// TIA Portal V18 export
FUNCTION "Status" : Void   // FC27, LAD
{ S7_Optimized_Access := 'TRUE' }
VERSION : 0.1
// stored: AutoNumber true, IsIECCheckEnabled false, SetENOAutomatically false, UDAEnableTagReadback false
BEGIN

REGION Network 1: Drive control A nok
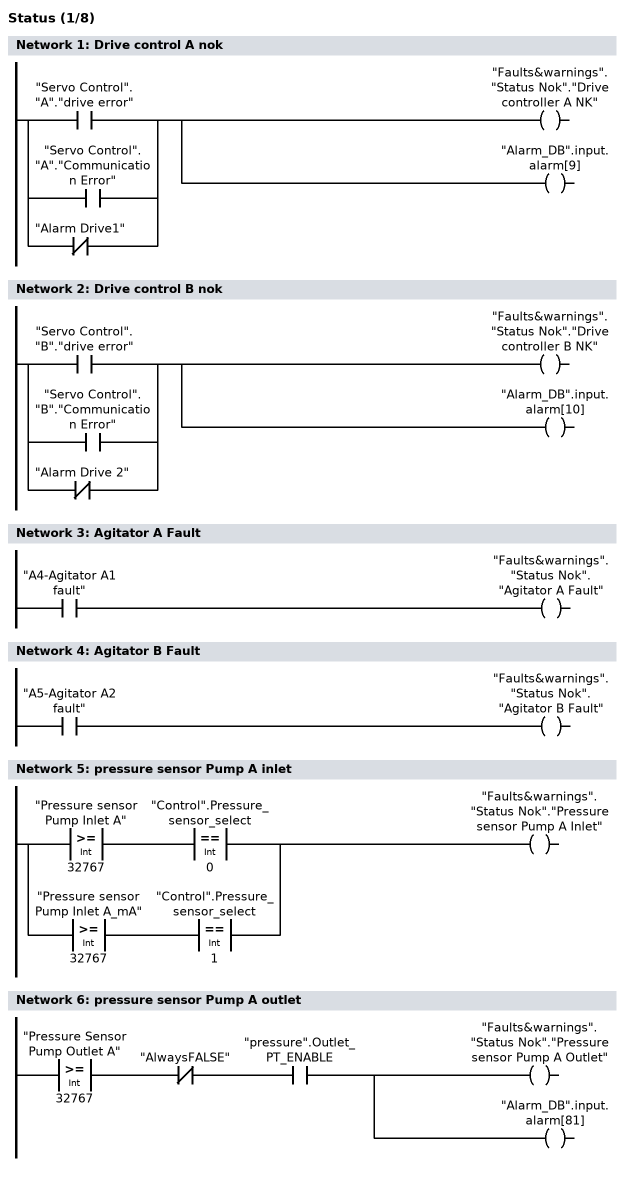
   RUNG wire#powerrail
      Contact( "Servo Control"."A"."drive error" )
      wire#w1
      Coil( "Faults&warnings"."Status Nok"."Drive controller A NK" )
   END_RUNG
   RUNG wire#powerrail
      Contact( "Servo Control"."A"."Communication Error" )
   END_RUNG wire#w1
   RUNG wire#powerrail
      I_Contact( "Alarm Drive1" )
   END_RUNG wire#w1
   RUNG wire#w1
      Coil( "Alarm_DB".input.alarm[9] )
   END_RUNG
   // the same network as SCL:
   "Faults&warnings"."Status Nok"."Drive controller A NK" := "Servo Control"."A"."drive error" OR "Servo Control"."A"."Communication Error" OR NOT "Alarm Drive1";
   "Alarm_DB".input.alarm[9] := "Faults&warnings"."Status Nok"."Drive controller A NK";
END_REGION

REGION Network 2: Drive control B nok
   RUNG wire#powerrail
      Contact( "Servo Control"."B"."drive error" )
      wire#w1
      Coil( "Faults&warnings"."Status Nok"."Drive controller B NK" )
   END_RUNG
   RUNG wire#powerrail
      Contact( "Servo Control"."B"."Communication Error" )
   END_RUNG wire#w1
   RUNG wire#powerrail
      I_Contact( "Alarm Drive 2" )
   END_RUNG wire#w1
   RUNG wire#w1
      Coil( "Alarm_DB".input.alarm[10] )
   END_RUNG
   // the same network as SCL:
   "Faults&warnings"."Status Nok"."Drive controller B NK" := "Servo Control"."B"."drive error" OR "Servo Control"."B"."Communication Error" OR NOT "Alarm Drive 2";
   "Alarm_DB".input.alarm[10] := "Faults&warnings"."Status Nok"."Drive controller B NK";
END_REGION

REGION Network 3: Agitator A Fault
   RUNG wire#powerrail
      Contact( "A4-Agitator A1 fault" )
      Coil( "Faults&warnings"."Status Nok"."Agitator A Fault" )
   END_RUNG
   // the same network as SCL:
   "Faults&warnings"."Status Nok"."Agitator A Fault" := "A4-Agitator A1 fault";
END_REGION

REGION Network 4: Agitator B Fault
   RUNG wire#powerrail
      Contact( "A5-Agitator A2 fault" )
      Coil( "Faults&warnings"."Status Nok"."Agitator B Fault" )
   END_RUNG
   // the same network as SCL:
   "Faults&warnings"."Status Nok"."Agitator B Fault" := "A5-Agitator A2 fault";
END_REGION

REGION Network 5: pressure sensor Pump A inlet
   RUNG wire#powerrail
      { S7_Templates := "SrcType := Int" } GE_Contact(in1 := "Pressure sensor Pump Inlet A", in2 := 32767)
      { S7_Templates := "SrcType := Int" } EQ_Contact(in1 := "Control".Pressure_sensor_select, in2 := 0)
      wire#w1
      Coil( "Faults&warnings"."Status Nok"."Pressure sensor Pump A Inlet" )
   END_RUNG
   RUNG wire#powerrail
      { S7_Templates := "SrcType := Int" } GE_Contact(in1 := "Pressure sensor Pump Inlet A_mA", in2 := 32767)
      { S7_Templates := "SrcType := Int" } EQ_Contact(in1 := "Control".Pressure_sensor_select, in2 := 1)
   END_RUNG wire#w1
   // the same network as SCL:
   "Faults&warnings"."Status Nok"."Pressure sensor Pump A Inlet" := (("Pressure sensor Pump Inlet A" >= 32767) AND ("Control".Pressure_sensor_select = 0)) OR (("Pressure sensor Pump Inlet A_mA" >= 32767) AND ("Control".Pressure_sensor_select = 1));
END_REGION

REGION Network 6: pressure sensor Pump A outlet
   RUNG wire#powerrail
      { S7_Templates := "SrcType := Int" } GE_Contact(in1 := "Pressure Sensor Pump Outlet A", in2 := 32767)
      I_Contact( "AlwaysFALSE" )
      Contact( "pressure".Outlet_PT_ENABLE )
      wire#w1
      Coil( "Faults&warnings"."Status Nok"."Pressure sensor Pump A Outlet" )
   END_RUNG
   RUNG wire#w1
      Coil( "Alarm_DB".input.alarm[81] )
   END_RUNG
   // the same network as SCL:
   "Faults&warnings"."Status Nok"."Pressure sensor Pump A Outlet" := ("Pressure Sensor Pump Outlet A" >= 32767) AND NOT "AlwaysFALSE" AND "pressure".Outlet_PT_ENABLE;
   "Alarm_DB".input.alarm[81] := "Faults&warnings"."Status Nok"."Pressure sensor Pump A Outlet";
END_REGION

REGION Network 7: pressure sensor Pump B inlet
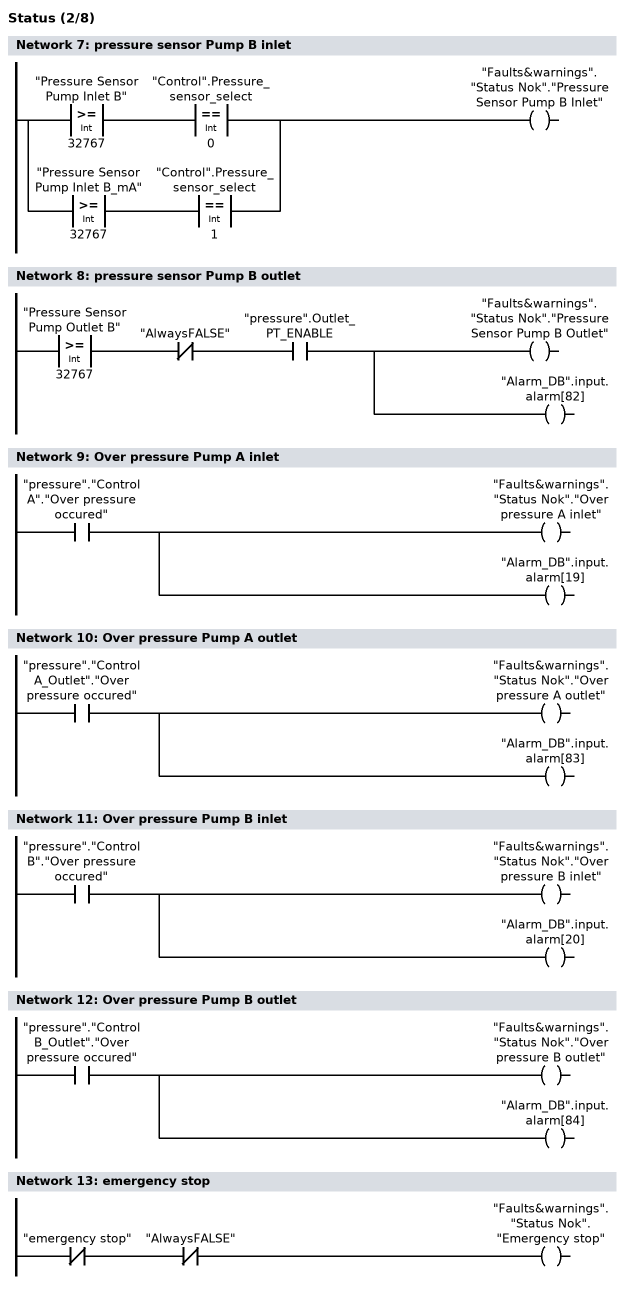
   RUNG wire#powerrail
      { S7_Templates := "SrcType := Int" } GE_Contact(in1 := "Pressure Sensor Pump Inlet B", in2 := 32767)
      { S7_Templates := "SrcType := Int" } EQ_Contact(in1 := "Control".Pressure_sensor_select, in2 := 0)
      wire#w1
      Coil( "Faults&warnings"."Status Nok"."Pressure Sensor Pump B Inlet" )
   END_RUNG
   RUNG wire#powerrail
      { S7_Templates := "SrcType := Int" } GE_Contact(in1 := "Pressure Sensor Pump Inlet B_mA", in2 := 32767)
      { S7_Templates := "SrcType := Int" } EQ_Contact(in1 := "Control".Pressure_sensor_select, in2 := 1)
   END_RUNG wire#w1
   // the same network as SCL:
   "Faults&warnings"."Status Nok"."Pressure Sensor Pump B Inlet" := (("Pressure Sensor Pump Inlet B" >= 32767) AND ("Control".Pressure_sensor_select = 0)) OR (("Pressure Sensor Pump Inlet B_mA" >= 32767) AND ("Control".Pressure_sensor_select = 1));
END_REGION

REGION Network 8: pressure sensor Pump B outlet
   RUNG wire#powerrail
      { S7_Templates := "SrcType := Int" } GE_Contact(in1 := "Pressure Sensor Pump Outlet B", in2 := 32767)
      I_Contact( "AlwaysFALSE" )
      Contact( "pressure".Outlet_PT_ENABLE )
      wire#w1
      Coil( "Faults&warnings"."Status Nok"."Pressure Sensor Pump B Outlet" )
   END_RUNG
   RUNG wire#w1
      Coil( "Alarm_DB".input.alarm[82] )
   END_RUNG
   // the same network as SCL:
   "Faults&warnings"."Status Nok"."Pressure Sensor Pump B Outlet" := ("Pressure Sensor Pump Outlet B" >= 32767) AND NOT "AlwaysFALSE" AND "pressure".Outlet_PT_ENABLE;
   "Alarm_DB".input.alarm[82] := "Faults&warnings"."Status Nok"."Pressure Sensor Pump B Outlet";
END_REGION

REGION Network 9: Over pressure Pump A inlet
   RUNG wire#powerrail
      Contact( "pressure"."Control A"."Over pressure occured" )
      wire#w1
      Coil( "Faults&warnings"."Status Nok"."Over pressure A inlet" )
   END_RUNG
   RUNG wire#w1
      Coil( "Alarm_DB".input.alarm[19] )
   END_RUNG
   // the same network as SCL:
   "Faults&warnings"."Status Nok"."Over pressure A inlet" := "pressure"."Control A"."Over pressure occured";
   "Alarm_DB".input.alarm[19] := "pressure"."Control A"."Over pressure occured";
END_REGION

REGION Network 10: Over pressure Pump A outlet
   RUNG wire#powerrail
      Contact( "pressure"."Control A_Outlet"."Over pressure occured" )
      wire#w1
      Coil( "Faults&warnings"."Status Nok"."Over pressure A outlet" )
   END_RUNG
   RUNG wire#w1
      Coil( "Alarm_DB".input.alarm[83] )
   END_RUNG
   // the same network as SCL:
   "Faults&warnings"."Status Nok"."Over pressure A outlet" := "pressure"."Control A_Outlet"."Over pressure occured";
   "Alarm_DB".input.alarm[83] := "pressure"."Control A_Outlet"."Over pressure occured";
END_REGION

REGION Network 11: Over pressure Pump B inlet
   RUNG wire#powerrail
      Contact( "pressure"."Control B"."Over pressure occured" )
      wire#w1
      Coil( "Faults&warnings"."Status Nok"."Over pressure B inlet" )
   END_RUNG
   RUNG wire#w1
      Coil( "Alarm_DB".input.alarm[20] )
   END_RUNG
   // the same network as SCL:
   "Faults&warnings"."Status Nok"."Over pressure B inlet" := "pressure"."Control B"."Over pressure occured";
   "Alarm_DB".input.alarm[20] := "pressure"."Control B"."Over pressure occured";
END_REGION

REGION Network 12: Over pressure Pump B outlet
   RUNG wire#powerrail
      Contact( "pressure"."Control B_Outlet"."Over pressure occured" )
      wire#w1
      Coil( "Faults&warnings"."Status Nok"."Over pressure B outlet" )
   END_RUNG
   RUNG wire#w1
      Coil( "Alarm_DB".input.alarm[84] )
   END_RUNG
   // the same network as SCL:
   "Faults&warnings"."Status Nok"."Over pressure B outlet" := "pressure"."Control B_Outlet"."Over pressure occured";
   "Alarm_DB".input.alarm[84] := "pressure"."Control B_Outlet"."Over pressure occured";
END_REGION

REGION Network 13: emergency stop
   RUNG wire#powerrail
      I_Contact( "emergency stop" )
      I_Contact( "AlwaysFALSE" )
      Coil( "Faults&warnings"."Status Nok"."Emergency stop" )
   END_RUNG
   // the same network as SCL:
   "Faults&warnings"."Status Nok"."Emergency stop" := NOT "emergency stop" AND NOT "AlwaysFALSE";
END_REGION

REGION Network 14: HEATER OK
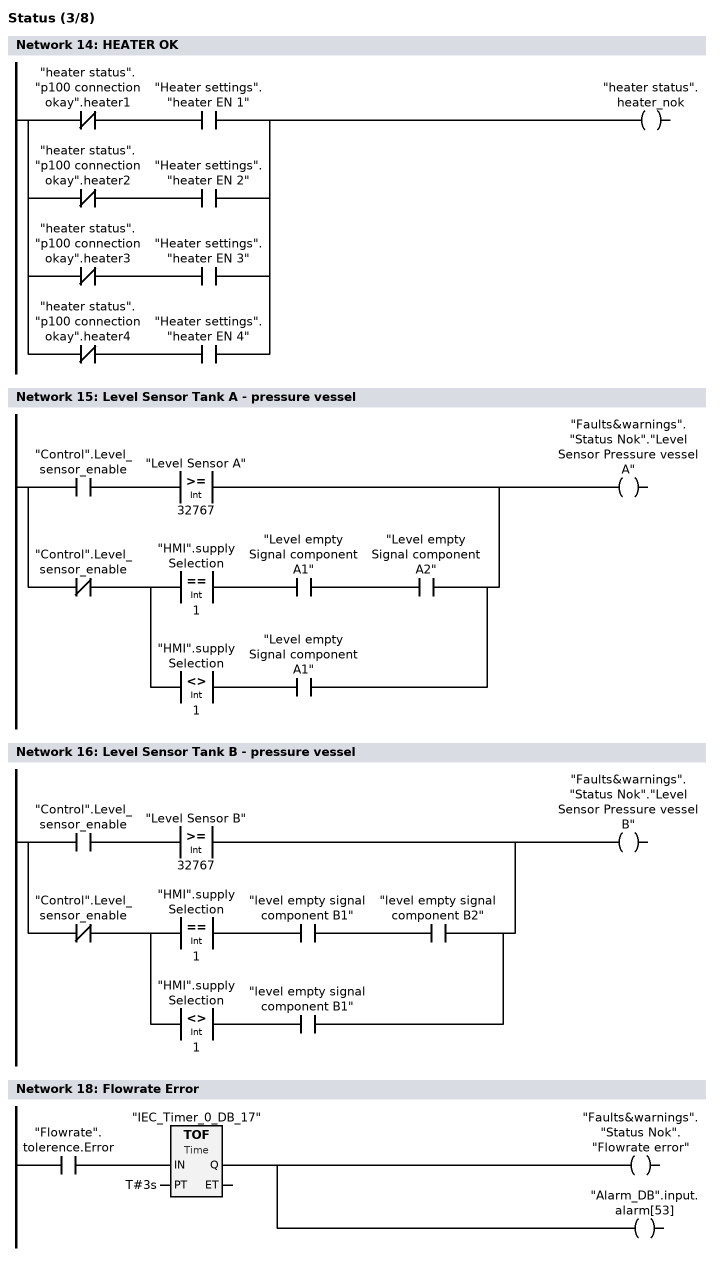
   RUNG wire#powerrail
      I_Contact( "heater status"."p100 connection okay".heater1 )
      Contact( "Heater settings"."heater EN 1" )
      wire#w1
      Coil( "heater status".heater_nok )
   END_RUNG
   RUNG wire#powerrail
      I_Contact( "heater status"."p100 connection okay".heater2 )
      Contact( "Heater settings"."heater EN 2" )
   END_RUNG wire#w1
   RUNG wire#powerrail
      I_Contact( "heater status"."p100 connection okay".heater3 )
      Contact( "Heater settings"."heater EN 3" )
   END_RUNG wire#w1
   RUNG wire#powerrail
      I_Contact( "heater status"."p100 connection okay".heater4 )
      Contact( "Heater settings"."heater EN 4" )
   END_RUNG wire#w1
   // the same network as SCL:
   "heater status".heater_nok := (NOT "heater status"."p100 connection okay".heater1 AND "Heater settings"."heater EN 1") OR (NOT "heater status"."p100 connection okay".heater2 AND "Heater settings"."heater EN 2") OR (NOT "heater status"."p100 connection okay".heater3 AND "Heater settings"."heater EN 3") OR (NOT "heater status"."p100 connection okay".heater4 AND "Heater settings"."heater EN 4");
END_REGION

REGION Network 15: Level Sensor Tank A - pressure vessel
   RUNG wire#powerrail
      Contact( "Control".Level_sensor_enable )
      { S7_Templates := "SrcType := Int" } GE_Contact(in1 := "Level Sensor A", in2 := 32767)
      wire#w1
      Coil( "Faults&warnings"."Status Nok"."Level Sensor Pressure vessel A" )
   END_RUNG
   RUNG wire#powerrail
      I_Contact( "Control".Level_sensor_enable )
      wire#w2
      { S7_Templates := "SrcType := Int" } EQ_Contact(in1 := "HMI".supplySelection, in2 := 1)
      Contact( "Level empty Signal component A1" )
      Contact( "Level empty Signal component A2" )
   END_RUNG wire#w1
   RUNG wire#w2
      { S7_Templates := "SrcType := Int" } NE_Contact(in1 := "HMI".supplySelection, in2 := 1)
      Contact( "Level empty Signal component A1" )
   END_RUNG wire#w1
   // the same network as SCL:
   "Faults&warnings"."Status Nok"."Level Sensor Pressure vessel A" := ("Control".Level_sensor_enable AND ("Level Sensor A" >= 32767)) OR (NOT "Control".Level_sensor_enable AND ((("HMI".supplySelection = 1) AND "Level empty Signal component A1" AND "Level empty Signal component A2") OR (("HMI".supplySelection <> 1) AND "Level empty Signal component A1")));
END_REGION

REGION Network 16: Level Sensor Tank B - pressure vessel
   RUNG wire#powerrail
      Contact( "Control".Level_sensor_enable )
      { S7_Templates := "SrcType := Int" } GE_Contact(in1 := "Level Sensor B", in2 := 32767)
      wire#w1
      Coil( "Faults&warnings"."Status Nok"."Level Sensor Pressure vessel B" )
   END_RUNG
   RUNG wire#powerrail
      I_Contact( "Control".Level_sensor_enable )
      wire#w2
      { S7_Templates := "SrcType := Int" } EQ_Contact(in1 := "HMI".supplySelection, in2 := 1)
      Contact( "level empty signal component B1" )
      Contact( "level empty signal component B2" )
   END_RUNG wire#w1
   RUNG wire#w2
      { S7_Templates := "SrcType := Int" } NE_Contact(in1 := "HMI".supplySelection, in2 := 1)
      Contact( "level empty signal component B1" )
   END_RUNG wire#w1
   // the same network as SCL:
   "Faults&warnings"."Status Nok"."Level Sensor Pressure vessel B" := ("Control".Level_sensor_enable AND ("Level Sensor B" >= 32767)) OR (NOT "Control".Level_sensor_enable AND ((("HMI".supplySelection = 1) AND "level empty signal component B1" AND "level empty signal component B2") OR (("HMI".supplySelection <> 1) AND "level empty signal component B1")));
END_REGION

REGION Network 17 (SCL): low level and empty level non tandum
   "Alarm_DB".input.alarm[40] := "Faults&warnings"."Status Nok"."Low level A1"  := "level"."Low level occured A";
   "Alarm_DB".input.alarm[42] := "Faults&warnings"."Status Nok"."Low level B1" := "level"."Low level occured B";

   "Faults&warnings"."Status Nok"."Level empty A1" := "level"."Level Empty A";
   "Alarm_DB".input.alarm[21] := "Faults&warnings"."Status Nok"."Level empty A1" OR "Temp".bit20;
   "Faults&warnings"."Status Nok"."Level empty B1" := "level"."Level Empty B";
   "Alarm_DB".input.alarm[23] := "Faults&warnings"."Status Nok"."Level empty B1" OR "Temp".bit21;

   "Faults&warnings"."Status Nok"."Level Low Drum A1" := "level"."Drum Level Low A1" AND "HMI".supplySelection = 1;
   "Faults&warnings"."Status Nok"."Level Low Drum A2" := "level"."Drum Level Low A2" AND "HMI".supplySelection = 1;
   "Faults&warnings"."Status Nok"."Level Low Drum B1" := "level"."Drum Level Low B1" AND "HMI".supplySelection = 1;
   "Faults&warnings"."Status Nok"."Level Low Drum B2" := "level"."Drum Level Low B2" AND "HMI".supplySelection = 1;

   "Faults&warnings"."Status Nok"."Level Empty Drum A1" := "level"."Drum Level Empty A1" AND "HMI".supplySelection = 1;
   "Faults&warnings"."Status Nok"."Level Empty Drum A2" := "level"."Drum Level Empty A2" AND "HMI".supplySelection = 1;
   "Faults&warnings"."Status Nok"."Level Empty Drum B1" := "level"."Drum Level Empty B1" AND "HMI".supplySelection = 1;
   "Faults&warnings"."Status Nok"."Level Empty Drum B2" := "level"."Drum Level Empty B2" AND "HMI".supplySelection = 1;
END_REGION

REGION Network 18: Flowrate Error
   RUNG wire#powerrail
      Contact( "Flowrate".tolerence.Error )
      { S7_Templates := "time_type := Time" } "IEC_Timer_0_DB_17".TOF(pt := T#3s, et =>)
      wire#w1
      Coil( "Faults&warnings"."Status Nok"."Flowrate error" )
   END_RUNG
   RUNG wire#w1
      Coil( "Alarm_DB".input.alarm[53] )
   END_RUNG
   // the same network as SCL:
   "IEC_Timer_0_DB_17".TOF(IN := "Flowrate".tolerence.Error, PT := T#3s);
   "Faults&warnings"."Status Nok"."Flowrate error" := "IEC_Timer_0_DB_17".Q;
   "Alarm_DB".input.alarm[53] := "IEC_Timer_0_DB_17".Q;
END_REGION

REGION Network 19: Critical Fault stop A metering
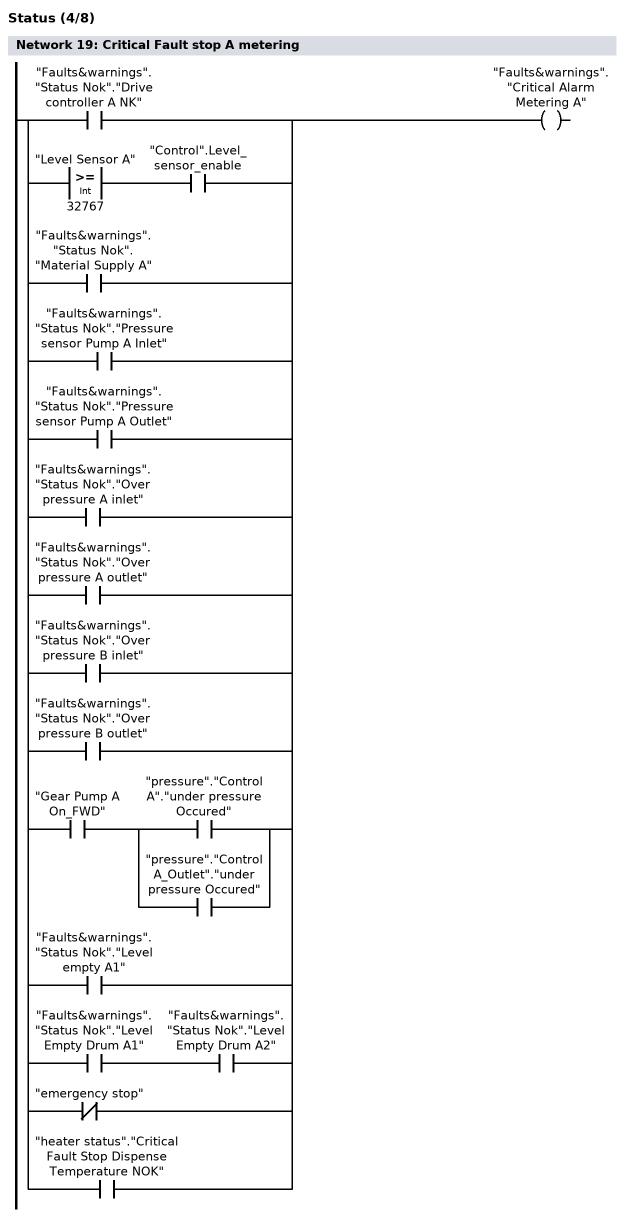
   RUNG wire#powerrail
      Contact( "Faults&warnings"."Status Nok"."Drive controller A NK" )
      wire#w1
      Coil( "Faults&warnings"."Critical Alarm Metering A" )
   END_RUNG
   RUNG wire#powerrail
      { S7_Templates := "SrcType := Int" } GE_Contact(in1 := "Level Sensor A", in2 := 32767)
      Contact( "Control".Level_sensor_enable )
   END_RUNG wire#w1
   RUNG wire#powerrail
      Contact( "Faults&warnings"."Status Nok"."Material Supply A" )
   END_RUNG wire#w1
   RUNG wire#powerrail
      Contact( "Faults&warnings"."Status Nok"."Pressure sensor Pump A Inlet" )
   END_RUNG wire#w1
   RUNG wire#powerrail
      Contact( "Faults&warnings"."Status Nok"."Pressure sensor Pump A Outlet" )
   END_RUNG wire#w1
   RUNG wire#powerrail
      Contact( "Faults&warnings"."Status Nok"."Over pressure A inlet" )
   END_RUNG wire#w1
   RUNG wire#powerrail
      Contact( "Faults&warnings"."Status Nok"."Over pressure A outlet" )
   END_RUNG wire#w1
   RUNG wire#powerrail
      Contact( "Faults&warnings"."Status Nok"."Over pressure B inlet" )
   END_RUNG wire#w1
   RUNG wire#powerrail
      Contact( "Faults&warnings"."Status Nok"."Over pressure B outlet" )
   END_RUNG wire#w1
   RUNG wire#powerrail
      Contact( "Gear Pump A On_FWD" )
      wire#w2
      Contact( "pressure"."Control A"."under pressure Occured" )
   END_RUNG wire#w1
   RUNG wire#w2
      Contact( "pressure"."Control A_Outlet"."under pressure Occured" )
   END_RUNG wire#w1
   RUNG wire#powerrail
      Contact( "Faults&warnings"."Status Nok"."Level empty A1" )
   END_RUNG wire#w1
   RUNG wire#powerrail
      Contact( "Faults&warnings"."Status Nok"."Level Empty Drum A1" )
      Contact( "Faults&warnings"."Status Nok"."Level Empty Drum A2" )
   END_RUNG wire#w1
   RUNG wire#powerrail
      I_Contact( "emergency stop" )
   END_RUNG wire#w1
   RUNG wire#powerrail
      Contact( "heater status"."Critical Fault Stop Dispense Temperature NOK" )
   END_RUNG wire#w1
   // the same network as SCL:
   "Faults&warnings"."Critical Alarm Metering A" := "Faults&warnings"."Status Nok"."Drive controller A NK" OR (("Level Sensor A" >= 32767) AND "Control".Level_sensor_enable) OR "Faults&warnings"."Status Nok"."Material Supply A" OR "Faults&warnings"."Status Nok"."Pressure sensor Pump A Inlet" OR "Faults&warnings"."Status Nok"."Pressure sensor Pump A Outlet" OR "Faults&warnings"."Status Nok"."Over pressure A inlet" OR "Faults&warnings"."Status Nok"."Over pressure A outlet" OR "Faults&warnings"."Status Nok"."Over pressure B inlet" OR "Faults&warnings"."Status Nok"."Over pressure B outlet" OR ("Gear Pump A On_FWD" AND ("pressure"."Control A"."under pressure Occured" OR "pressure"."Control A_Outlet"."under pressure Occured")) OR "Faults&warnings"."Status Nok"."Level empty A1" OR ("Faults&warnings"."Status Nok"."Level Empty Drum A1" AND "Faults&warnings"."Status Nok"."Level Empty Drum A2") OR NOT "emergency stop" OR "heater status"."Critical Fault Stop Dispense Temperature NOK";
END_REGION

REGION Network 20: Critical Fault stop B metering
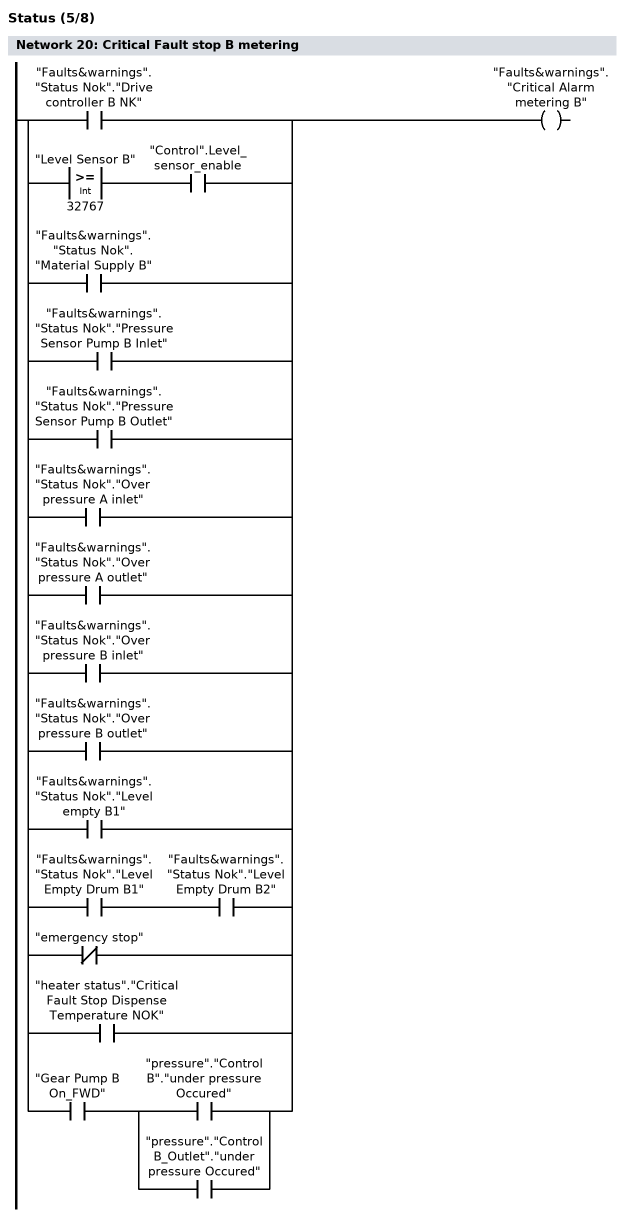
   RUNG wire#powerrail
      Contact( "Faults&warnings"."Status Nok"."Drive controller B NK" )
      wire#w1
      Coil( "Faults&warnings"."Critical Alarm metering B" )
   END_RUNG
   RUNG wire#powerrail
      { S7_Templates := "SrcType := Int" } GE_Contact(in1 := "Level Sensor B", in2 := 32767)
      Contact( "Control".Level_sensor_enable )
   END_RUNG wire#w1
   RUNG wire#powerrail
      Contact( "Faults&warnings"."Status Nok"."Material Supply B" )
   END_RUNG wire#w1
   RUNG wire#powerrail
      Contact( "Faults&warnings"."Status Nok"."Pressure Sensor Pump B Inlet" )
   END_RUNG wire#w1
   RUNG wire#powerrail
      Contact( "Faults&warnings"."Status Nok"."Pressure Sensor Pump B Outlet" )
   END_RUNG wire#w1
   RUNG wire#powerrail
      Contact( "Faults&warnings"."Status Nok"."Over pressure A inlet" )
   END_RUNG wire#w1
   RUNG wire#powerrail
      Contact( "Faults&warnings"."Status Nok"."Over pressure A outlet" )
   END_RUNG wire#w1
   RUNG wire#powerrail
      Contact( "Faults&warnings"."Status Nok"."Over pressure B inlet" )
   END_RUNG wire#w1
   RUNG wire#powerrail
      Contact( "Faults&warnings"."Status Nok"."Over pressure B outlet" )
   END_RUNG wire#w1
   RUNG wire#powerrail
      Contact( "Faults&warnings"."Status Nok"."Level empty B1" )
   END_RUNG wire#w1
   RUNG wire#powerrail
      Contact( "Faults&warnings"."Status Nok"."Level Empty Drum B1" )
      Contact( "Faults&warnings"."Status Nok"."Level Empty Drum B2" )
   END_RUNG wire#w1
   RUNG wire#powerrail
      I_Contact( "emergency stop" )
   END_RUNG wire#w1
   RUNG wire#powerrail
      Contact( "heater status"."Critical Fault Stop Dispense Temperature NOK" )
   END_RUNG wire#w1
   RUNG wire#powerrail
      Contact( "Gear Pump B On_FWD" )
      wire#w2
      Contact( "pressure"."Control B"."under pressure Occured" )
   END_RUNG wire#w1
   RUNG wire#w2
      Contact( "pressure"."Control B_Outlet"."under pressure Occured" )
   END_RUNG wire#w1
   // the same network as SCL:
   "Faults&warnings"."Critical Alarm metering B" := "Faults&warnings"."Status Nok"."Drive controller B NK" OR (("Level Sensor B" >= 32767) AND "Control".Level_sensor_enable) OR "Faults&warnings"."Status Nok"."Material Supply B" OR "Faults&warnings"."Status Nok"."Pressure Sensor Pump B Inlet" OR "Faults&warnings"."Status Nok"."Pressure Sensor Pump B Outlet" OR "Faults&warnings"."Status Nok"."Over pressure A inlet" OR "Faults&warnings"."Status Nok"."Over pressure A outlet" OR "Faults&warnings"."Status Nok"."Over pressure B inlet" OR "Faults&warnings"."Status Nok"."Over pressure B outlet" OR "Faults&warnings"."Status Nok"."Level empty B1" OR ("Faults&warnings"."Status Nok"."Level Empty Drum B1" AND "Faults&warnings"."Status Nok"."Level Empty Drum B2") OR NOT "emergency stop" OR "heater status"."Critical Fault Stop Dispense Temperature NOK" OR ("Gear Pump B On_FWD" AND ("pressure"."Control B"."under pressure Occured" OR "pressure"."Control B_Outlet"."under pressure Occured"));
END_REGION

REGION Network 21: critical alarm AB
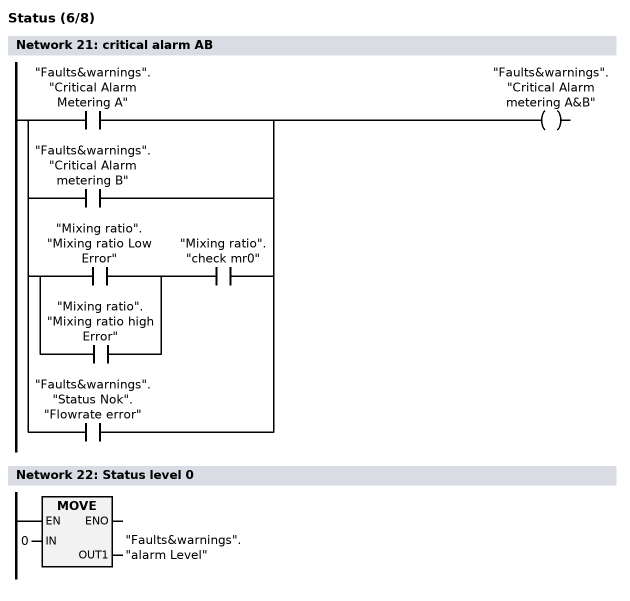
   RUNG wire#powerrail
      Contact( "Faults&warnings"."Critical Alarm Metering A" )
      wire#w1
      Coil( "Faults&warnings"."Critical Alarm metering A&B" )
   END_RUNG
   RUNG wire#powerrail
      Contact( "Faults&warnings"."Critical Alarm metering B" )
   END_RUNG wire#w1
   RUNG wire#powerrail
      Contact( "Mixing ratio"."Mixing ratio Low  Error" )
      wire#w2
      Contact( "Mixing ratio"."check mr0" )
   END_RUNG wire#w1
   RUNG wire#powerrail
      Contact( "Mixing ratio"."Mixing ratio high Error" )
   END_RUNG wire#w2
   RUNG wire#powerrail
      Contact( "Faults&warnings"."Status Nok"."Flowrate error" )
   END_RUNG wire#w1
   // the same network as SCL:
   "Faults&warnings"."Critical Alarm metering A&B" := "Faults&warnings"."Critical Alarm Metering A" OR "Faults&warnings"."Critical Alarm metering B" OR (("Mixing ratio"."Mixing ratio Low  Error" OR "Mixing ratio"."Mixing ratio high Error") AND "Mixing ratio"."check mr0") OR "Faults&warnings"."Status Nok"."Flowrate error";
END_REGION

REGION Network 22: Status level 0
   RUNG wire#powerrail
      Move(in := 0, out1 => "Faults&warnings"."alarm Level")
   END_RUNG
   // the same network as SCL:
   "Faults&warnings"."alarm Level" := 0;
END_REGION

REGION Network 23: Status level 1/warning
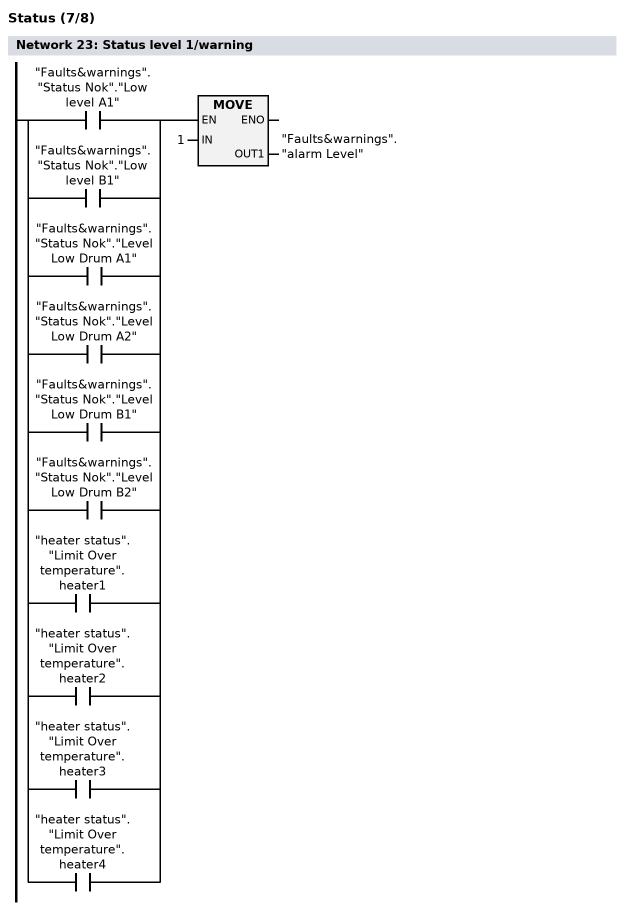
   RUNG wire#powerrail
      Contact( "Faults&warnings"."Status Nok"."Low level A1" )
      wire#w1
      Move(in := 1, out1 => "Faults&warnings"."alarm Level")
   END_RUNG
   RUNG wire#powerrail
      Contact( "Faults&warnings"."Status Nok"."Low level B1" )
   END_RUNG wire#w1
   RUNG wire#powerrail
      Contact( "Faults&warnings"."Status Nok"."Level Low Drum A1" )
   END_RUNG wire#w1
   RUNG wire#powerrail
      Contact( "Faults&warnings"."Status Nok"."Level Low Drum A2" )
   END_RUNG wire#w1
   RUNG wire#powerrail
      Contact( "Faults&warnings"."Status Nok"."Level Low Drum B1" )
   END_RUNG wire#w1
   RUNG wire#powerrail
      Contact( "Faults&warnings"."Status Nok"."Level Low Drum B2" )
   END_RUNG wire#w1
   RUNG wire#powerrail
      Contact( "heater status"."Limit Over temperature".heater1 )
   END_RUNG wire#w1
   RUNG wire#powerrail
      Contact( "heater status"."Limit Over temperature".heater2 )
   END_RUNG wire#w1
   RUNG wire#powerrail
      Contact( "heater status"."Limit Over temperature".heater3 )
   END_RUNG wire#w1
   RUNG wire#powerrail
      Contact( "heater status"."Limit Over temperature".heater4 )
   END_RUNG wire#w1
   // the same network as SCL:
   IF "Faults&warnings"."Status Nok"."Low level A1" OR "Faults&warnings"."Status Nok"."Low level B1" OR "Faults&warnings"."Status Nok"."Level Low Drum A1" OR "Faults&warnings"."Status Nok"."Level Low Drum A2" OR "Faults&warnings"."Status Nok"."Level Low Drum B1" OR "Faults&warnings"."Status Nok"."Level Low Drum B2" OR "heater status"."Limit Over temperature".heater1 OR "heater status"."Limit Over temperature".heater2 OR "heater status"."Limit Over temperature".heater3 OR "heater status"."Limit Over temperature".heater4 THEN
       "Faults&warnings"."alarm Level" := 1;
   END_IF;
END_REGION

REGION Network 24: Status level 1/fault
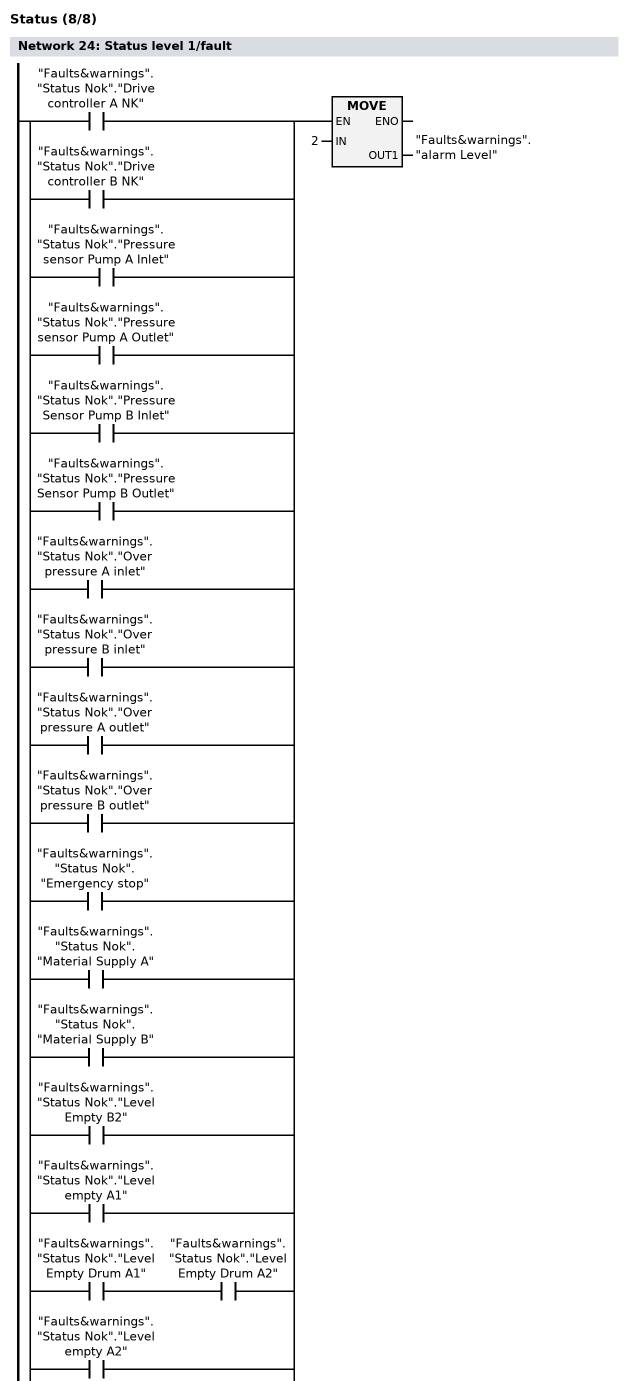
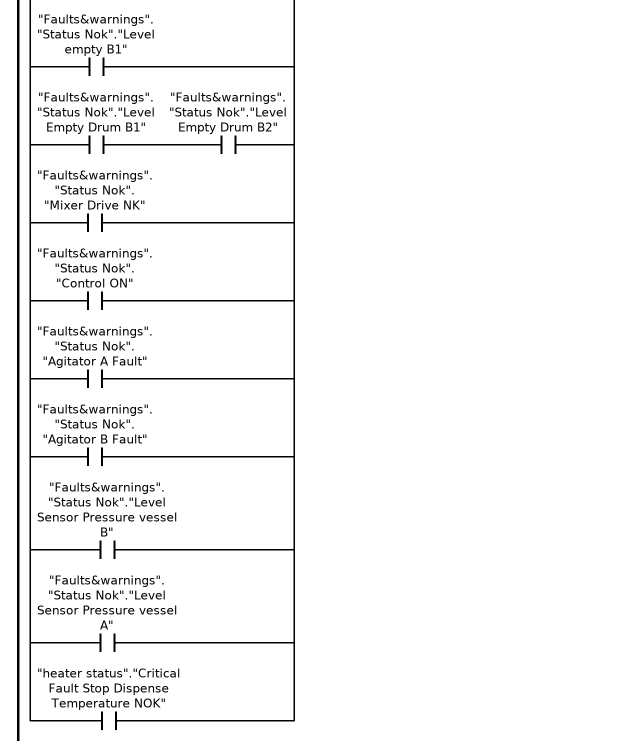
   RUNG wire#powerrail
      Contact( "Faults&warnings"."Status Nok"."Drive controller A NK" )
      wire#w1
      Move(in := 2, out1 => "Faults&warnings"."alarm Level")
   END_RUNG
   RUNG wire#powerrail
      Contact( "Faults&warnings"."Status Nok"."Drive controller B NK" )
   END_RUNG wire#w1
   RUNG wire#powerrail
      Contact( "Faults&warnings"."Status Nok"."Pressure sensor Pump A Inlet" )
   END_RUNG wire#w1
   RUNG wire#powerrail
      Contact( "Faults&warnings"."Status Nok"."Pressure sensor Pump A Outlet" )
   END_RUNG wire#w1
   RUNG wire#powerrail
      Contact( "Faults&warnings"."Status Nok"."Pressure Sensor Pump B Inlet" )
   END_RUNG wire#w1
   RUNG wire#powerrail
      Contact( "Faults&warnings"."Status Nok"."Pressure Sensor Pump B Outlet" )
   END_RUNG wire#w1
   RUNG wire#powerrail
      Contact( "Faults&warnings"."Status Nok"."Over pressure A inlet" )
   END_RUNG wire#w1
   RUNG wire#powerrail
      Contact( "Faults&warnings"."Status Nok"."Over pressure B inlet" )
   END_RUNG wire#w1
   RUNG wire#powerrail
      Contact( "Faults&warnings"."Status Nok"."Over pressure A outlet" )
   END_RUNG wire#w1
   RUNG wire#powerrail
      Contact( "Faults&warnings"."Status Nok"."Over pressure B outlet" )
   END_RUNG wire#w1
   RUNG wire#powerrail
      Contact( "Faults&warnings"."Status Nok"."Emergency stop" )
   END_RUNG wire#w1
   RUNG wire#powerrail
      Contact( "Faults&warnings"."Status Nok"."Material Supply A" )
   END_RUNG wire#w1
   RUNG wire#powerrail
      Contact( "Faults&warnings"."Status Nok"."Material Supply B" )
   END_RUNG wire#w1
   RUNG wire#powerrail
      Contact( "Faults&warnings"."Status Nok"."Level Empty B2" )
   END_RUNG wire#w1
   RUNG wire#powerrail
      Contact( "Faults&warnings"."Status Nok"."Level empty A1" )
   END_RUNG wire#w1
   RUNG wire#powerrail
      Contact( "Faults&warnings"."Status Nok"."Level Empty Drum A1" )
      Contact( "Faults&warnings"."Status Nok"."Level Empty Drum A2" )
   END_RUNG wire#w1
   RUNG wire#powerrail
      Contact( "Faults&warnings"."Status Nok"."Level empty A2" )
   END_RUNG wire#w1
   RUNG wire#powerrail
      Contact( "Faults&warnings"."Status Nok"."Level empty B1" )
   END_RUNG wire#w1
   RUNG wire#powerrail
      Contact( "Faults&warnings"."Status Nok"."Level Empty Drum B1" )
      Contact( "Faults&warnings"."Status Nok"."Level Empty Drum B2" )
   END_RUNG wire#w1
   RUNG wire#powerrail
      Contact( "Faults&warnings"."Status Nok"."Mixer Drive NK" )
   END_RUNG wire#w1
   RUNG wire#powerrail
      Contact( "Faults&warnings"."Status Nok"."Control ON" )
   END_RUNG wire#w1
   RUNG wire#powerrail
      Contact( "Faults&warnings"."Status Nok"."Agitator A Fault" )
   END_RUNG wire#w1
   RUNG wire#powerrail
      Contact( "Faults&warnings"."Status Nok"."Agitator B Fault" )
   END_RUNG wire#w1
   RUNG wire#powerrail
      Contact( "Faults&warnings"."Status Nok"."Level Sensor Pressure vessel B" )
   END_RUNG wire#w1
   RUNG wire#powerrail
      Contact( "Faults&warnings"."Status Nok"."Level Sensor Pressure vessel A" )
   END_RUNG wire#w1
   RUNG wire#powerrail
      Contact( "heater status"."Critical Fault Stop Dispense Temperature NOK" )
   END_RUNG wire#w1
   // the same network as SCL:
   IF "Faults&warnings"."Status Nok"."Drive controller A NK" OR "Faults&warnings"."Status Nok"."Drive controller B NK" OR "Faults&warnings"."Status Nok"."Pressure sensor Pump A Inlet" OR "Faults&warnings"."Status Nok"."Pressure sensor Pump A Outlet" OR "Faults&warnings"."Status Nok"."Pressure Sensor Pump B Inlet" OR "Faults&warnings"."Status Nok"."Pressure Sensor Pump B Outlet" OR "Faults&warnings"."Status Nok"."Over pressure A inlet" OR "Faults&warnings"."Status Nok"."Over pressure B inlet" OR "Faults&warnings"."Status Nok"."Over pressure A outlet" OR "Faults&warnings"."Status Nok"."Over pressure B outlet" OR "Faults&warnings"."Status Nok"."Emergency stop" OR "Faults&warnings"."Status Nok"."Material Supply A" OR "Faults&warnings"."Status Nok"."Material Supply B" OR "Faults&warnings"."Status Nok"."Level Empty B2" OR "Faults&warnings"."Status Nok"."Level empty A1" OR ("Faults&warnings"."Status Nok"."Level Empty Drum A1" AND "Faults&warnings"."Status Nok"."Level Empty Drum A2") OR "Faults&warnings"."Status Nok"."Level empty A2" OR "Faults&warnings"."Status Nok"."Level empty B1" OR ("Faults&warnings"."Status Nok"."Level Empty Drum B1" AND "Faults&warnings"."Status Nok"."Level Empty Drum B2") OR "Faults&warnings"."Status Nok"."Mixer Drive NK" OR "Faults&warnings"."Status Nok"."Control ON" OR "Faults&warnings"."Status Nok"."Agitator A Fault" OR "Faults&warnings"."Status Nok"."Agitator B Fault" OR "Faults&warnings"."Status Nok"."Level Sensor Pressure vessel B" OR "Faults&warnings"."Status Nok"."Level Sensor Pressure vessel A" OR "heater status"."Critical Fault Stop Dispense Temperature NOK" THEN
       "Faults&warnings"."alarm Level" := 2;
   END_IF;
END_REGION
END_FUNCTION
